// TIA Portal project "0001_v19_pulseGenerator" (V19)

(* hardware
DEVICE "S7-1200 station_1"  S7-1200 Station
   slot 0: "Rack_0"  S7-1200 Rack  Rack  V1.0
   slot 1: "PLC_1"  CPU 1212C DC/DC/DC  6ES7 212-1AE40-0XB0  V4.6
*)

// ===== PLC "PLC_1"  CPU 1212C DC/DC/DC =====

VAR_GLOBAL   // PLC tag table "Default tag table"
   "SWITCH" AT %I0.0 : Bool;
   "OUTPUT" AT %Q0.0 : Bool;
END_VAR

VAR_GLOBAL   // PLC tag table "Tag table_1"
   "PUSH BUTTON" AT %M0.1 : Bool;
   "PUSH BUTTON MEMORY" AT %M0.2 : Bool;
   "PULSE MEMORY" AT %M0.3 : Bool;
END_VAR

// folder: System blocks/Program resources

DATA_BLOCK "IEC_Timer_0_DB"   // DB1
{ S7_Optimized_Access := 'TRUE' }
AUTHOR : Simatic
FAMILY : IEC
NAME : IEC_TMR
VERSION : 1.0
// stored: InstanceOfName IEC_TIMER
"IEC_TIMER"
BEGIN
END_DATA_BLOCK

DATA_BLOCK "IEC_Timer_0_DB_1"   // DB2
{ S7_Optimized_Access := 'TRUE' }
AUTHOR : Simatic
FAMILY : IEC
NAME : IEC_TMR
VERSION : 1.0
// stored: InstanceOfName IEC_TIMER
"IEC_TIMER"
BEGIN
END_DATA_BLOCK

DATA_BLOCK "IEC_Timer_0_DB_2"   // DB3
{ S7_Optimized_Access := 'TRUE' }
AUTHOR : Simatic
FAMILY : IEC
NAME : IEC_TMR
VERSION : 1.0
// stored: InstanceOfName IEC_TIMER
"IEC_TIMER"
BEGIN
END_DATA_BLOCK

// folder: (top level)

ORGANIZATION_BLOCK "Main"   // OB1, LAD, ProgramCycle
TITLE = "Main Program Sweep (Cycle)"
{ S7_Optimized_Access := 'TRUE' }
VERSION : 0.1
   VAR_INPUT
      Initial_Call : Bool;   // Initial call of this OB
      Remanence : Bool;   // =True, if remanent data are available
   END_VAR
   VAR_TEMP   // added for the SCL form of the ladder/FBD networks
      _w1 : Bool;
   END_VAR
BEGIN

REGION Network 1
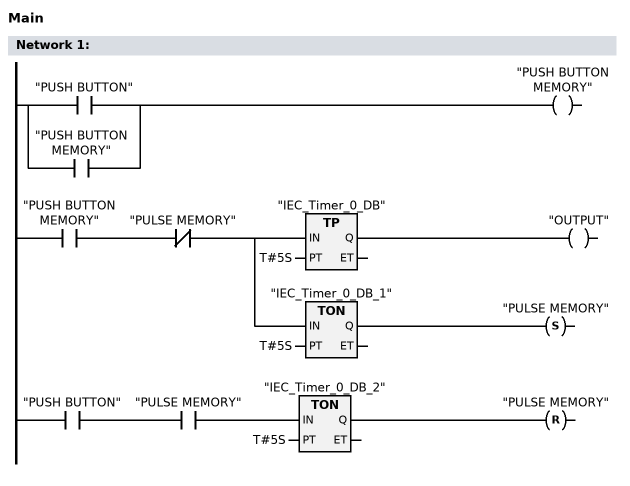
   "PUSH BUTTON MEMORY" := "PUSH BUTTON" OR "PUSH BUTTON MEMORY";
   #_w1 := "PUSH BUTTON MEMORY" AND NOT "PULSE MEMORY";
   "IEC_Timer_0_DB".TP(IN := #_w1, PT := T#5S);
   "OUTPUT" := "IEC_Timer_0_DB".Q;
   "IEC_Timer_0_DB_1".TON(IN := #_w1, PT := T#5S);
   IF "IEC_Timer_0_DB_1".Q THEN "PULSE MEMORY" := TRUE; END_IF;
   "IEC_Timer_0_DB_2".TON(IN := "PUSH BUTTON" AND "PULSE MEMORY", PT := T#5S);
   IF "IEC_Timer_0_DB_2".Q THEN "PULSE MEMORY" := FALSE; END_IF;
END_REGION
END_ORGANIZATION_BLOCK